// Mitsubishi GX Works2 project: Powder Spray robot1+ServoN   PLC: Q03UDV
// 20181022A

// task MAIN (event TRUE, interval 0, priority 31): MAIN
// task MAIN1 (event TRUE, interval 0, priority 31): MAIN1_Block000, MAIN1_Block001, MAIN1_Block002
// task OFS (event TRUE, interval 0, priority 31): OFS
// task LIFTER (event TRUE, interval 0, priority 31): LIFTER
// task 64AD (event TRUE, interval 0, priority 31): 64AD
// task SERVO (event TRUE, interval 0, priority 31): SERVO
// task D62 (event TRUE, interval 0, priority 31): D62
// task POWDER1 (event TRUE, interval 0, priority 31): POWDER1
// task POWDER2 (event TRUE, interval 0, priority 31): POWDER2
// task 62DA (event TRUE, interval 0, priority 31): 62DA

PROGRAM MAIN
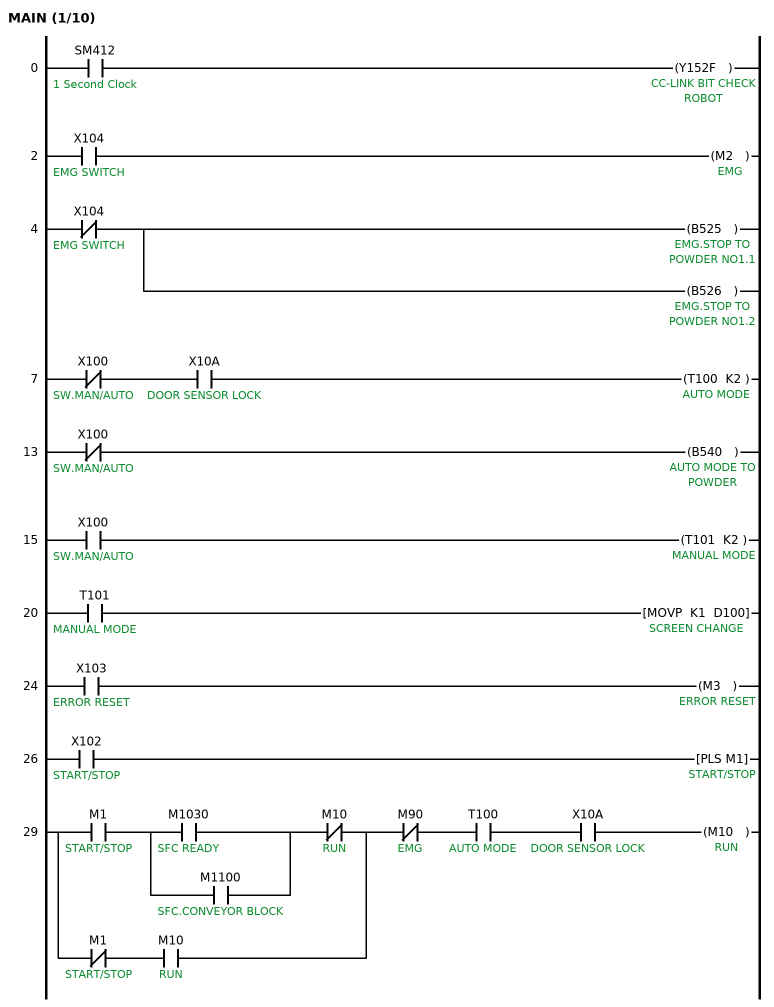
0     LD      SM412  ; 1 Second Clock
      OUT     Y152F  ; CC-LINK BIT CHECK ROBOT
2     LD      X104  ; EMG SWITCH
      OUT     M2  ; EMG
4     LDI     X104  ; EMG SWITCH
      OUT     B525  ; EMG.STOP TO POWDER NO1.1
      OUT     B526  ; EMG.STOP TO POWDER NO1.2
7     LDI     X100  ; SW.MAN/AUTO
      AND     X10A  ; DOOR SENSOR LOCK
      OUT     T100 K2  ; AUTO MODE
13    LDI     X100  ; SW.MAN/AUTO
      OUT     B540  ; AUTO MODE TO POWDER
15    LD      X100  ; SW.MAN/AUTO
      OUT     T101 K2  ; MANUAL MODE
20    LD      T101  ; MANUAL MODE
      MOVP    K1 D100  ; SCREEN CHANGE
24    LD      X103  ; ERROR RESET
      OUT     M3  ; ERROR RESET
26    LD      X102  ; START/STOP
      PLS     M1  ; START/STOP
29    LD      M1  ; START/STOP
      LD      M1030  ; SFC READY
      OR      M1100  ; SFC.CONVEYOR BLOCK
      ANB
      ANI     M10  ; RUN
      LDI     M1  ; START/STOP
      AND     M10  ; RUN
      ORB
      ANI     M90  ; EMG
      AND     T100  ; AUTO MODE
      AND     X10A  ; DOOR SENSOR LOCK
      OUT     M10  ; RUN
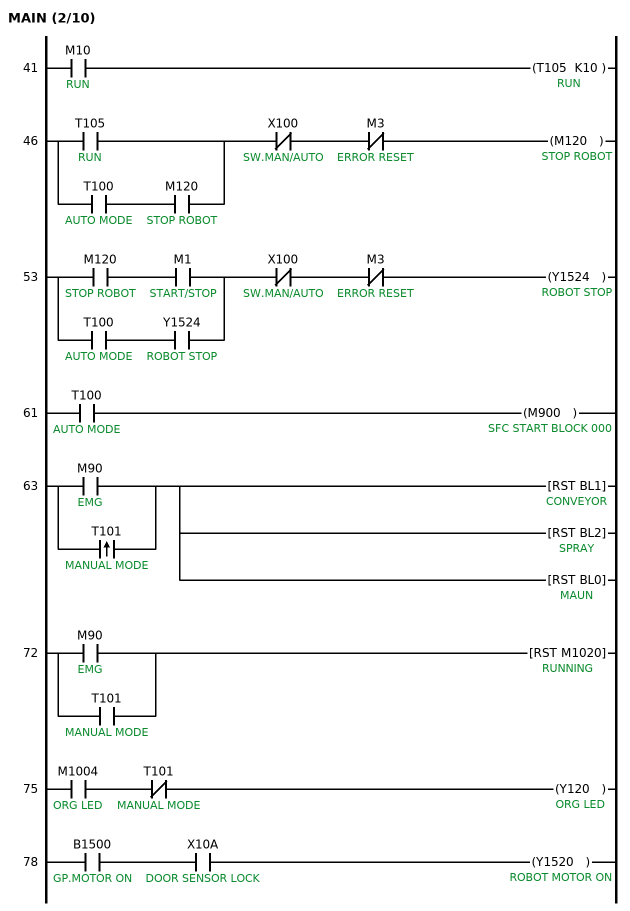
41    LD      M10  ; RUN
      OUT     T105 K10  ; RUN
46    LD      T105  ; RUN
      LD      T100  ; AUTO MODE
      AND     M120  ; STOP ROBOT
      ORB
      ANI     X100  ; SW.MAN/AUTO
      ANI     M3  ; ERROR RESET
      OUT     M120  ; STOP ROBOT
53    LD      M120  ; STOP ROBOT
      AND     M1  ; START/STOP
      LD      T100  ; AUTO MODE
      AND     Y1524  ; ROBOT STOP
      ORB
      ANI     X100  ; SW.MAN/AUTO
      ANI     M3  ; ERROR RESET
      OUT     Y1524  ; ROBOT STOP
61    LD      T100  ; AUTO MODE
      OUT     M900  ; SFC START BLOCK 000
63    LD      M90  ; EMG
      ORP     T101  ; MANUAL MODE
      RST     BL1  ; CONVEYOR
      RST     BL2  ; SPRAY
      RST     BL0  ; MAUN
72    LD      M90  ; EMG
      OR      T101  ; MANUAL MODE
      RST     M1020  ; RUNNING
75    LD      M1004  ; ORG LED
      ANI     T101  ; MANUAL MODE
      OUT     Y120  ; ORG LED
78    LD      B1500  ; GP.MOTOR ON
      AND     X10A  ; DOOR SENSOR LOCK
      OUT     Y1520  ; ROBOT MOTOR ON
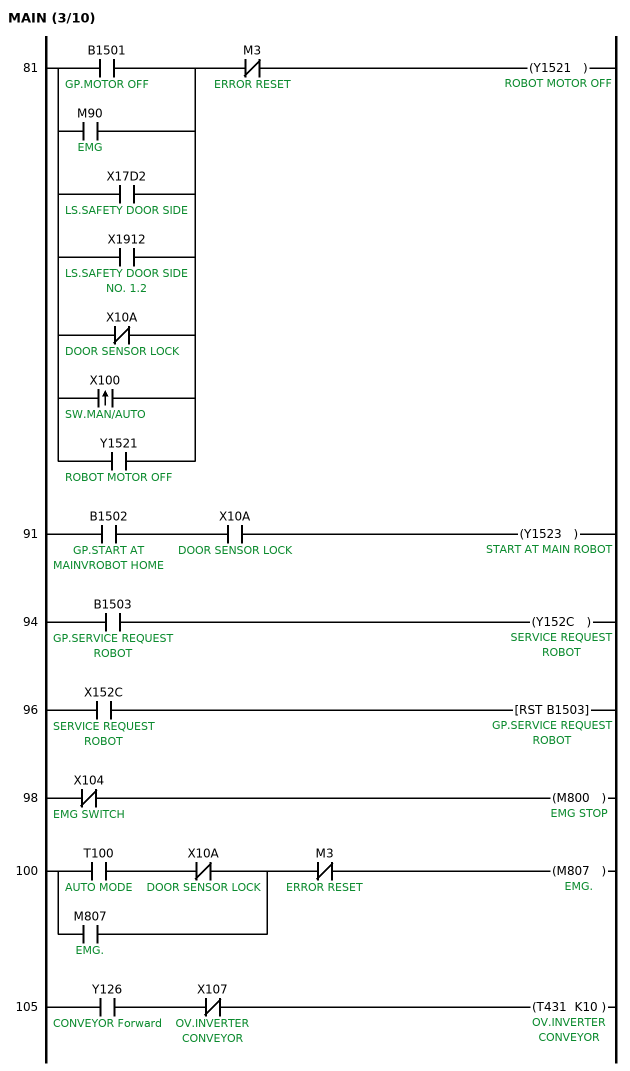
81    LD      B1501  ; GP.MOTOR OFF
      OR      M90  ; EMG
      OR      X17D2  ; LS.SAFETY DOOR SIDE
      OR      X1912  ; LS.SAFETY DOOR SIDE NO. 1.2
      ORI     X10A  ; DOOR SENSOR LOCK
      ORP     X100  ; SW.MAN/AUTO
      OR      Y1521  ; ROBOT MOTOR OFF
      ANI     M3  ; ERROR RESET
      OUT     Y1521  ; ROBOT MOTOR OFF
91    LD      B1502  ; GP.START AT MAINVROBOT HOME
      AND     X10A  ; DOOR SENSOR LOCK
      OUT     Y1523  ; START AT MAIN ROBOT
94    LD      B1503  ; GP.SERVICE REQUEST ROBOT
      OUT     Y152C  ; SERVICE REQUEST ROBOT
96    LD      X152C  ; SERVICE REQUEST ROBOT
      RST     B1503  ; GP.SERVICE REQUEST ROBOT
98    LDI     X104  ; EMG SWITCH
      OUT     M800  ; EMG STOP
100   LD      T100  ; AUTO MODE
      ANI     X10A  ; DOOR SENSOR LOCK
      OR      M807  ; EMG.
      ANI     M3  ; ERROR RESET
      OUT     M807  ; EMG.
105   LD      Y126  ; CONVEYOR Forward
      ANI     X107  ; OV.INVERTER CONVEYOR
      OUT     T431 K10  ; OV.INVERTER CONVEYOR
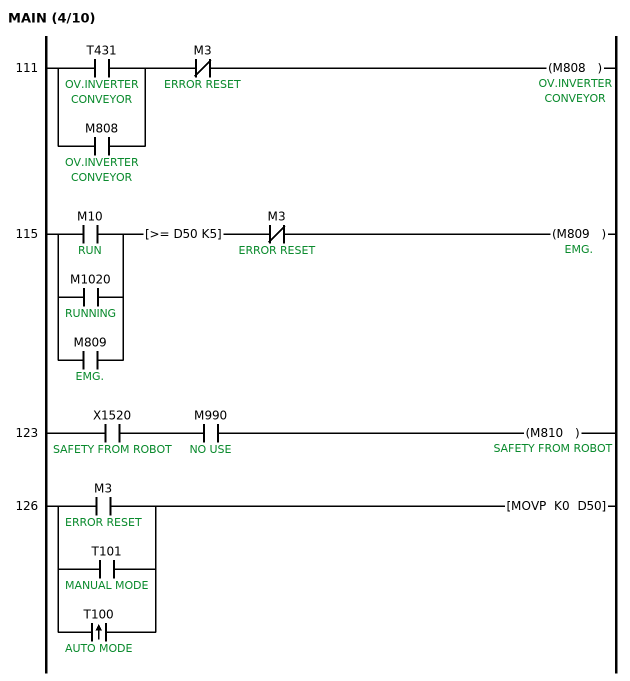
111   LD      T431  ; OV.INVERTER CONVEYOR
      OR      M808  ; OV.INVERTER CONVEYOR
      ANI     M3  ; ERROR RESET
      OUT     M808  ; OV.INVERTER CONVEYOR
115   LD      M10  ; RUN
      OR      M1020  ; RUNNING
      OR      M809  ; EMG.
      AND>=   D50 K5
      ANI     M3  ; ERROR RESET
      OUT     M809  ; EMG.
123   LD      X1520  ; SAFETY FROM ROBOT
      AND     M990  ; NO USE
      OUT     M810  ; SAFETY FROM ROBOT
126   LD      M3  ; ERROR RESET
      OR      T101  ; MANUAL MODE
      ORP     T100  ; AUTO MODE
      MOVP    K0 D50
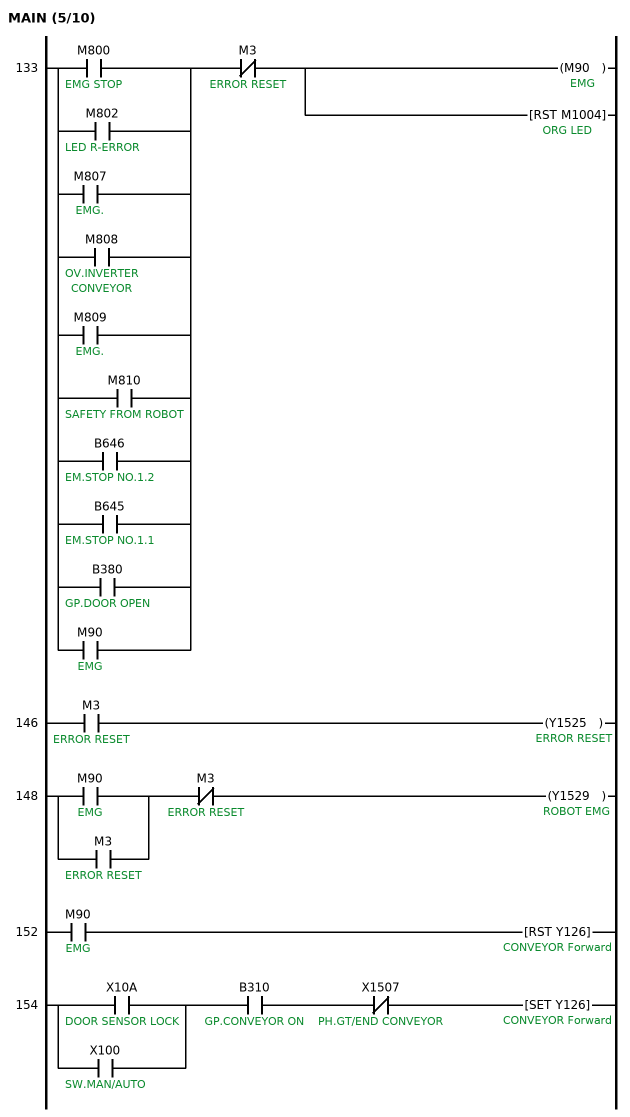
133   LD      M800  ; EMG STOP
      OR      M802  ; LED R-ERROR
      OR      M807  ; EMG.
      OR      M808  ; OV.INVERTER CONVEYOR
      OR      M809  ; EMG.
      OR      M810  ; SAFETY FROM ROBOT
      OR      B646  ; EM.STOP NO.1.2
      OR      B645  ; EM.STOP NO.1.1
      OR      B380  ; GP.DOOR OPEN
      OR      M90  ; EMG
      ANI     M3  ; ERROR RESET
      OUT     M90  ; EMG
      RST     M1004  ; ORG LED
146   LD      M3  ; ERROR RESET
      OUT     Y1525  ; ERROR RESET
148   LD      M90  ; EMG
      OR      M3  ; ERROR RESET
      ANI     M3  ; ERROR RESET
      OUT     Y1529  ; ROBOT EMG
152   LD      M90  ; EMG
      RST     Y126  ; CONVEYOR Forward
154   LD      X10A  ; DOOR SENSOR LOCK
      OR      X100  ; SW.MAN/AUTO
      AND     B310  ; GP.CONVEYOR ON
      ANI     X1507  ; PH.GT/END CONVEYOR
      SET     Y126  ; CONVEYOR Forward
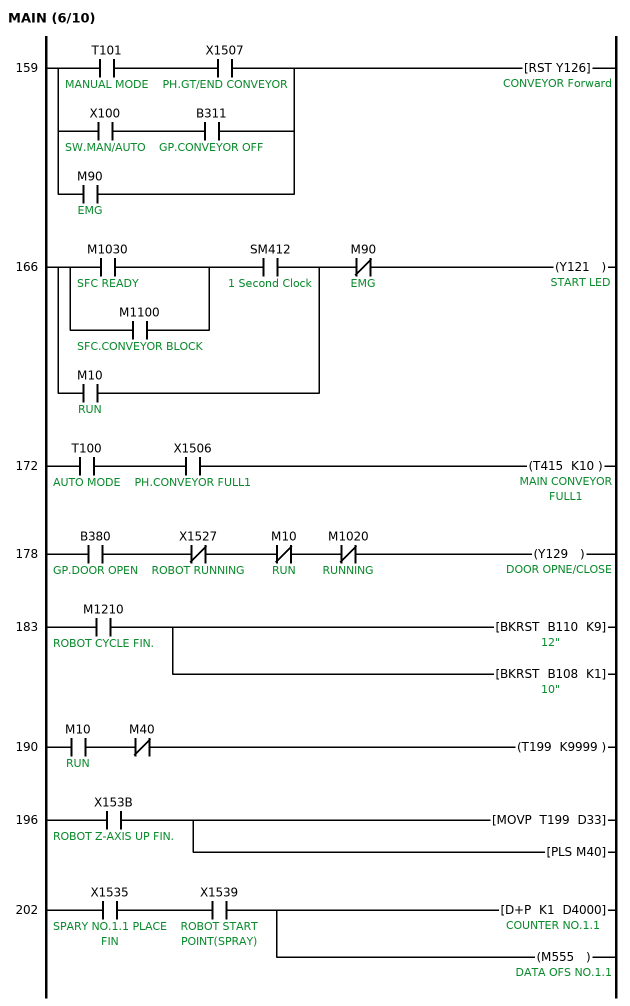
159   LD      T101  ; MANUAL MODE
      AND     X1507  ; PH.GT/END CONVEYOR
      LD      X100  ; SW.MAN/AUTO
      AND     B311  ; GP.CONVEYOR OFF
      ORB
      OR      M90  ; EMG
      RST     Y126  ; CONVEYOR Forward
166   LD      M1030  ; SFC READY
      OR      M1100  ; SFC.CONVEYOR BLOCK
      AND     SM412  ; 1 Second Clock
      OR      M10  ; RUN
      ANI     M90  ; EMG
      OUT     Y121  ; START LED
172   LD      T100  ; AUTO MODE
      AND     X1506  ; PH.CONVEYOR FULL1
      OUT     T415 K10  ; MAIN CONVEYOR FULL1
178   LD      B380  ; GP.DOOR OPEN
      ANI     X1527  ; ROBOT RUNNING
      ANI     M10  ; RUN
      ANI     M1020  ; RUNNING
      OUT     Y129  ; DOOR OPNE/CLOSE
183   LD      M1210  ; ROBOT CYCLE FIN.
      BKRST   B110 K9  ; 12"
      BKRST   B108 K1  ; 10"
190   LD      M10  ; RUN
      ANI     M40
      OUT     T199 K9999
196   LD      X153B  ; ROBOT Z-AXIS UP FIN.
      MOVP    T199 D33
      PLS     M40
202   LD      X1535  ; SPARY NO.1.1 PLACE FIN
      AND     X1539  ; ROBOT START POINT(SPRAY)
      D+P     K1 D4000  ; COUNTER NO.1.1
      OUT     M555  ; DATA OFS NO.1.1
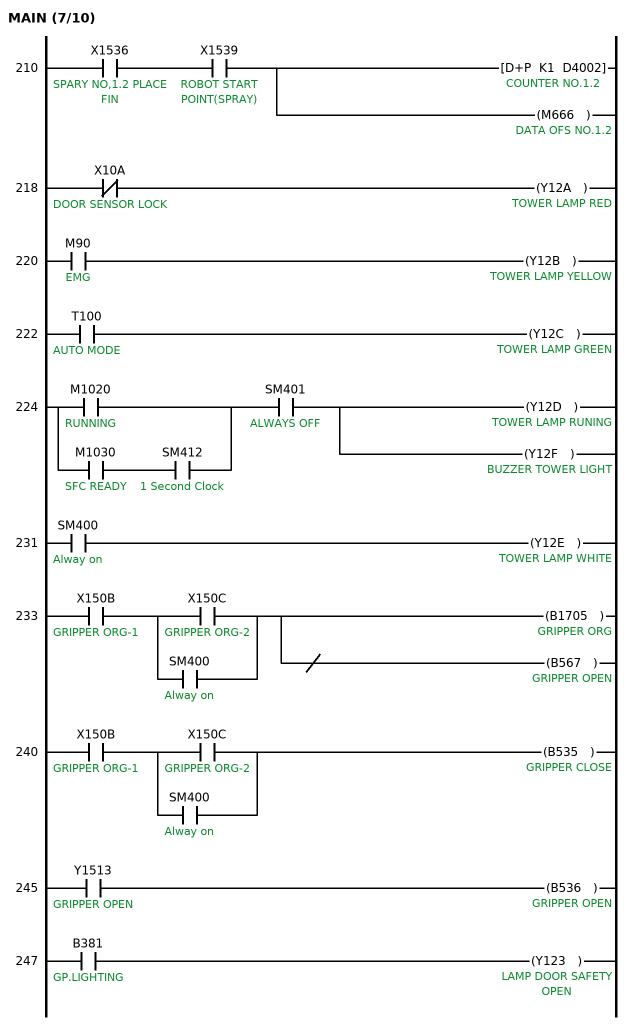
210   LD      X1536  ; SPARY NO,1.2 PLACE FIN
      AND     X1539  ; ROBOT START POINT(SPRAY)
      D+P     K1 D4002  ; COUNTER NO.1.2
      OUT     M666  ; DATA OFS NO.1.2
218   LDI     X10A  ; DOOR SENSOR LOCK
      OUT     Y12A  ; TOWER LAMP RED
220   LD      M90  ; EMG
      OUT     Y12B  ; TOWER LAMP YELLOW
222   LD      T100  ; AUTO MODE
      OUT     Y12C  ; TOWER LAMP GREEN
224   LD      M1020  ; RUNNING
      LD      M1030  ; SFC READY
      AND     SM412  ; 1 Second Clock
      ORB
      AND     SM401  ; ALWAYS OFF
      OUT     Y12D  ; TOWER LAMP RUNING
      OUT     Y12F  ; BUZZER TOWER LIGHT
231   LD      SM400  ; Alway on
      OUT     Y12E  ; TOWER LAMP WHITE
233   LD      X150B  ; GRIPPER ORG-1
      LD      X150C  ; GRIPPER ORG-2
      OR      SM400  ; Alway on
      ANB
      OUT     B1705  ; GRIPPER ORG
      INV
      OUT     B567  ; GRIPPER OPEN
240   LD      X150B  ; GRIPPER ORG-1
      LD      X150C  ; GRIPPER ORG-2
      OR      SM400  ; Alway on
      ANB
      OUT     B535  ; GRIPPER CLOSE
245   LD      Y1513  ; GRIPPER OPEN
      OUT     B536  ; GRIPPER OPEN
247   LD      B381  ; GP.LIGHTING
      OUT     Y123  ; LAMP DOOR SAFETY OPEN
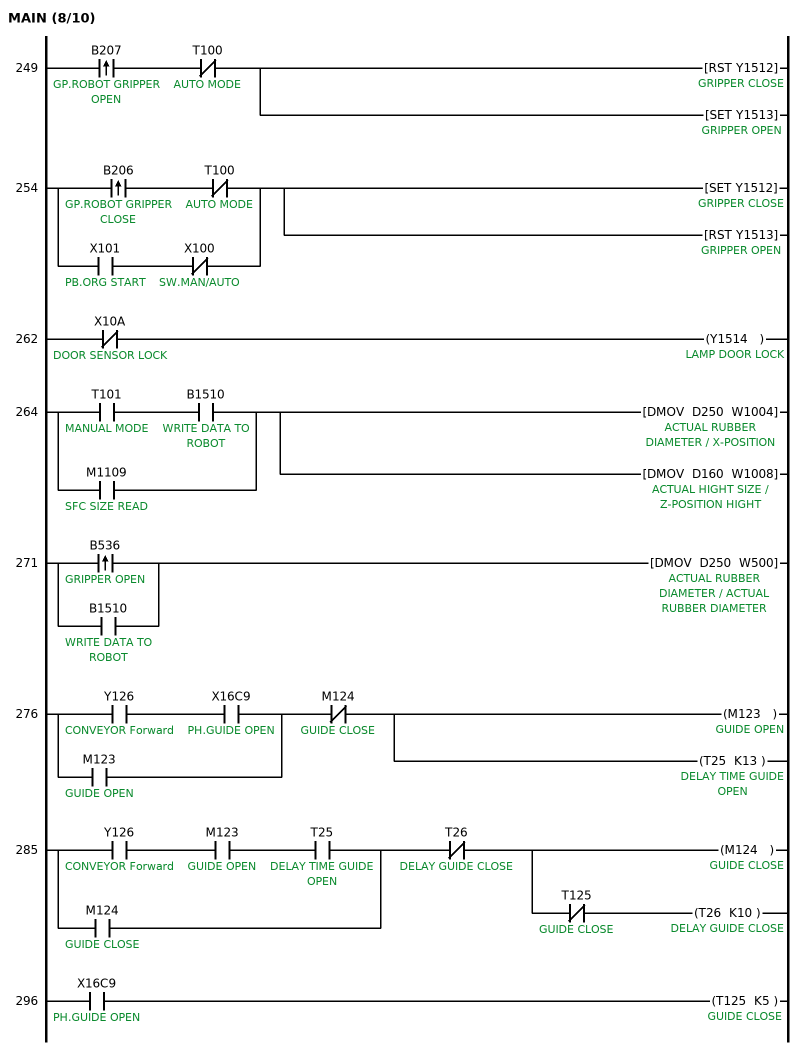
249   LDP     B207  ; GP.ROBOT GRIPPER OPEN
      ANI     T100  ; AUTO MODE
      RST     Y1512  ; GRIPPER CLOSE
      SET     Y1513  ; GRIPPER OPEN
254   LDP     B206  ; GP.ROBOT GRIPPER CLOSE
      ANI     T100  ; AUTO MODE
      LD      X101  ; PB.ORG START
      ANI     X100  ; SW.MAN/AUTO
      ORB
      SET     Y1512  ; GRIPPER CLOSE
      RST     Y1513  ; GRIPPER OPEN
262   LDI     X10A  ; DOOR SENSOR LOCK
      OUT     Y1514  ; LAMP DOOR LOCK
264   LD      T101  ; MANUAL MODE
      AND     B1510  ; WRITE DATA TO ROBOT
      OR      M1109  ; SFC SIZE READ
      DMOV    D250 W1004  ; ACTUAL RUBBER DIAMETER / X-POSITION
      DMOV    D160 W1008  ; ACTUAL HIGHT SIZE / Z-POSITION HIGHT
271   LDP     B536  ; GRIPPER OPEN
      OR      B1510  ; WRITE DATA TO ROBOT
      DMOV    D250 W500  ; ACTUAL RUBBER DIAMETER
276   LD      Y126  ; CONVEYOR Forward
      AND     X16C9  ; PH.GUIDE OPEN
      OR      M123  ; GUIDE OPEN
      ANI     M124  ; GUIDE CLOSE
      OUT     M123  ; GUIDE OPEN
      OUT     T25 K13  ; DELAY TIME GUIDE OPEN
285   LD      Y126  ; CONVEYOR Forward
      AND     M123  ; GUIDE OPEN
      AND     T25  ; DELAY TIME GUIDE OPEN
      OR      M124  ; GUIDE CLOSE
      ANI     T26  ; DELAY GUIDE CLOSE
      OUT     M124  ; GUIDE CLOSE
      ANI     T125  ; GUIDE CLOSE
      OUT     T26 K10  ; DELAY GUIDE CLOSE
296   LD      X16C9  ; PH.GUIDE OPEN
      OUT     T125 K5  ; GUIDE CLOSE
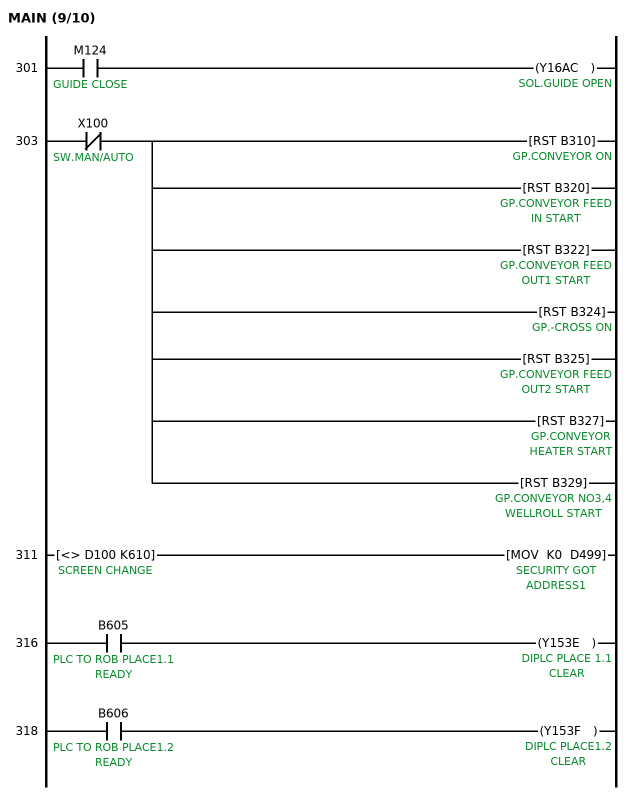
301   LD      M124  ; GUIDE CLOSE
      OUT     Y16AC  ; SOL.GUIDE OPEN
303   LDI     X100  ; SW.MAN/AUTO
      RST     B310  ; GP.CONVEYOR ON
      RST     B320  ; GP.CONVEYOR FEED IN START
      RST     B322  ; GP.CONVEYOR FEED OUT1 START
      RST     B324  ; GP.-CROSS ON
      RST     B325  ; GP.CONVEYOR FEED OUT2 START
      RST     B327  ; GP.CONVEYOR HEATER START
      RST     B329  ; GP.CONVEYOR NO3,4 WELLROLL START
311   LD<>    D100 K610  ; SCREEN CHANGE
      MOV     K0 D499  ; SECURITY GOT ADDRESS1
316   LD      B605  ; PLC TO ROB PLACE1.1 READY
      OUT     Y153E  ; DIPLC PLACE 1.1 CLEAR
318   LD      B606  ; PLC TO ROB PLACE1.2 READY
      OUT     Y153F  ; DIPLC PLACE1.2  CLEAR
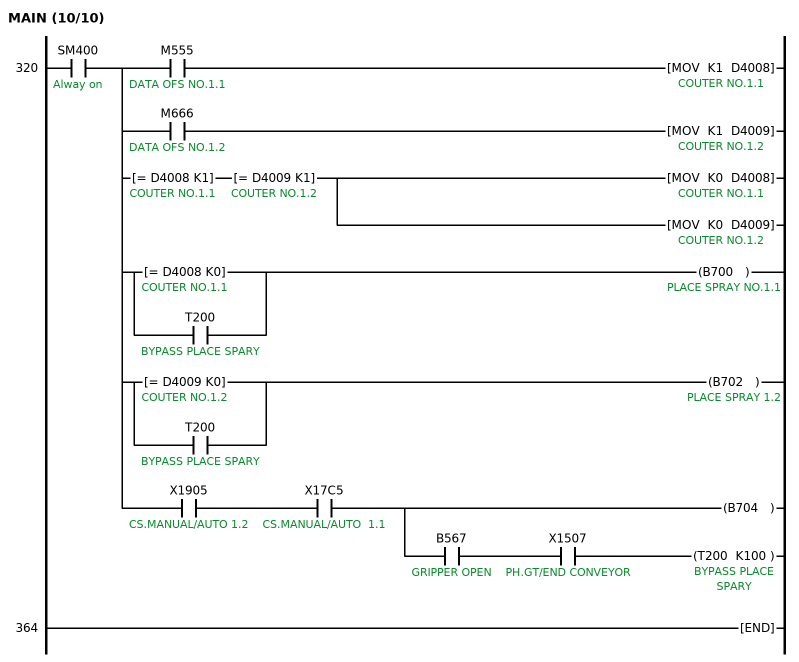
320   LD      SM400  ; Alway on
      MPS
      AND     M555  ; DATA OFS NO.1.1
      MOV     K1 D4008  ; COUTER NO.1.1
      MRD
      AND     M666  ; DATA OFS NO.1.2
      MOV     K1 D4009  ; COUTER NO.1.2
      MRD
      AND=    D4008 K1  ; COUTER NO.1.1
      AND=    D4009 K1  ; COUTER NO.1.2
      MOV     K0 D4008
      MOV     K0 D4009
      MRD
      LD=     D4008 K0  ; COUTER NO.1.1
      OR      T200  ; BYPASS PLACE SPARY
      ANB
      OUT     B700  ; PLACE SPRAY NO.1.1
      MRD
      LD=     D4009 K0  ; COUTER NO.1.2
      OR      T200  ; BYPASS PLACE SPARY
      ANB
      OUT     B702  ; PLACE SPRAY 1.2
      MPP
      AND     X1905  ; CS.MANUAL/AUTO 1.2
      AND     X17C5  ; CS.MANUAL/AUTO  1.1
      OUT     B704
      AND     B567  ; GRIPPER OPEN
      AND     X1507  ; PH.GT/END CONVEYOR
      OUT     T200 K100  ; BYPASS PLACE SPARY
364   END
END_PROGRAM

PROGRAM OFS
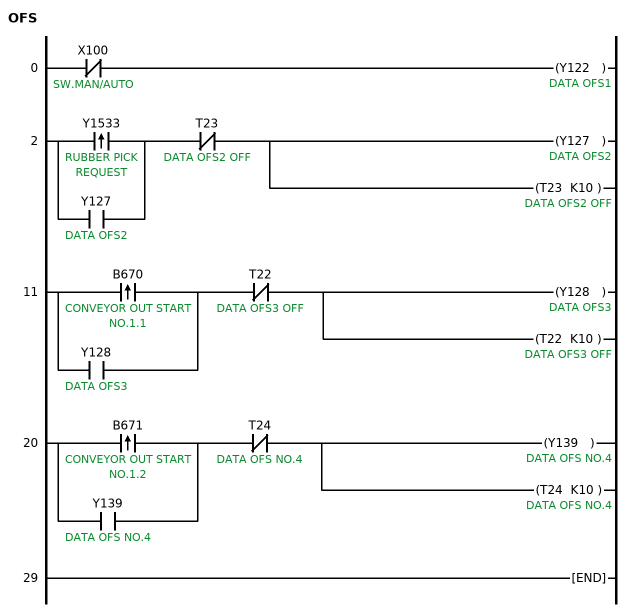
0     LDI     X100  ; SW.MAN/AUTO
      OUT     Y122  ; DATA OFS1
2     LDP     Y1533  ; RUBBER PICK  REQUEST
      OR      Y127  ; DATA OFS2
      ANI     T23  ; DATA OFS2 OFF
      OUT     Y127  ; DATA OFS2
      OUT     T23 K10  ; DATA OFS2 OFF
11    LDP     B670  ; CONVEYOR OUT START NO.1.1
      OR      Y128  ; DATA OFS3
      ANI     T22  ; DATA OFS3 OFF
      OUT     Y128  ; DATA OFS3
      OUT     T22 K10  ; DATA OFS3 OFF
20    LDP     B671  ; CONVEYOR OUT START NO.1.2
      OR      Y139  ; DATA OFS NO.4
      ANI     T24  ; DATA OFS NO.4
      OUT     Y139  ; DATA OFS NO.4
      OUT     T24 K10  ; DATA OFS NO.4
29    END
END_PROGRAM

PROGRAM LIFTER
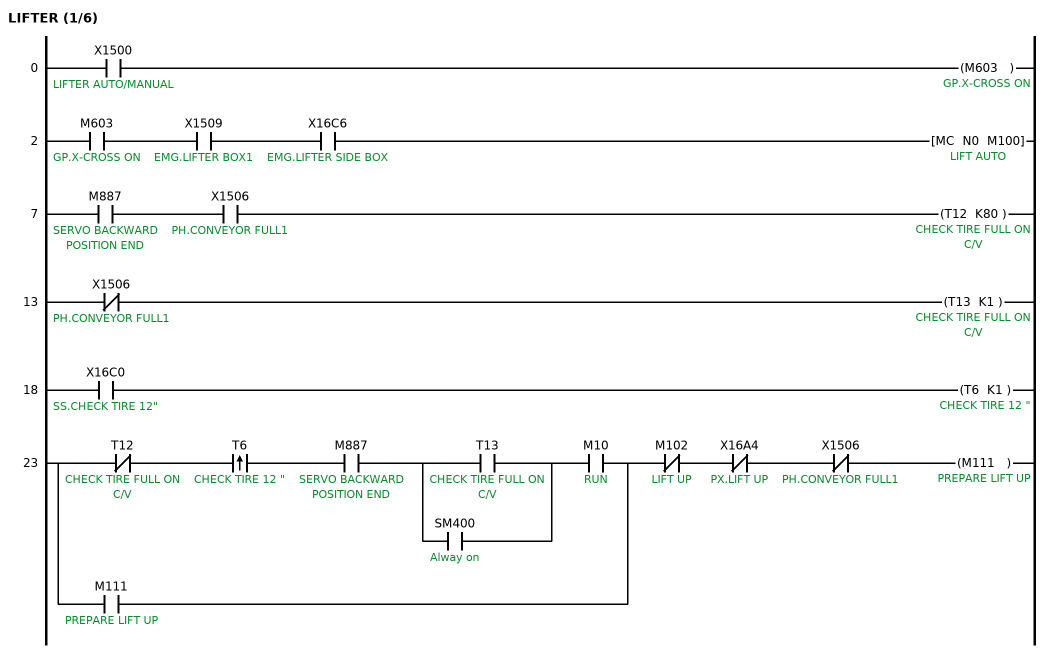
0     LD      X1500  ; LIFTER AUTO/MANUAL
      OUT     M603  ; GP.X-CROSS ON
2     LD      M603  ; GP.X-CROSS ON
      AND     X1509  ; EMG.LIFTER BOX1
      AND     X16C6  ; EMG.LIFTER SIDE BOX
      MC      N0 M100  ; LIFT AUTO
7     LD      M887  ; SERVO BACKWARD POSITION END
      AND     X1506  ; PH.CONVEYOR FULL1
      OUT     T12 K80  ; CHECK TIRE FULL ON C/V
13    LDI     X1506  ; PH.CONVEYOR FULL1
      OUT     T13 K1  ; CHECK TIRE FULL ON C/V
18    LD      X16C0  ; SS.CHECK TIRE 12"
      OUT     T6 K1  ; CHECK TIRE 12 "
23    LDI     T12  ; CHECK TIRE FULL ON C/V
      ANDP    T6  ; CHECK TIRE 12 "
      AND     M887  ; SERVO BACKWARD POSITION END
      LD      T13  ; CHECK TIRE FULL ON C/V
      OR      SM400  ; Alway on
      ANB
      AND     M10  ; RUN
      OR      M111  ; PREPARE LIFT UP
      ANI     M102  ; LIFT UP
      ANI     X16A4  ; PX.LIFT UP
      ANI     X1506  ; PH.CONVEYOR FULL1
      OUT     M111  ; PREPARE LIFT UP
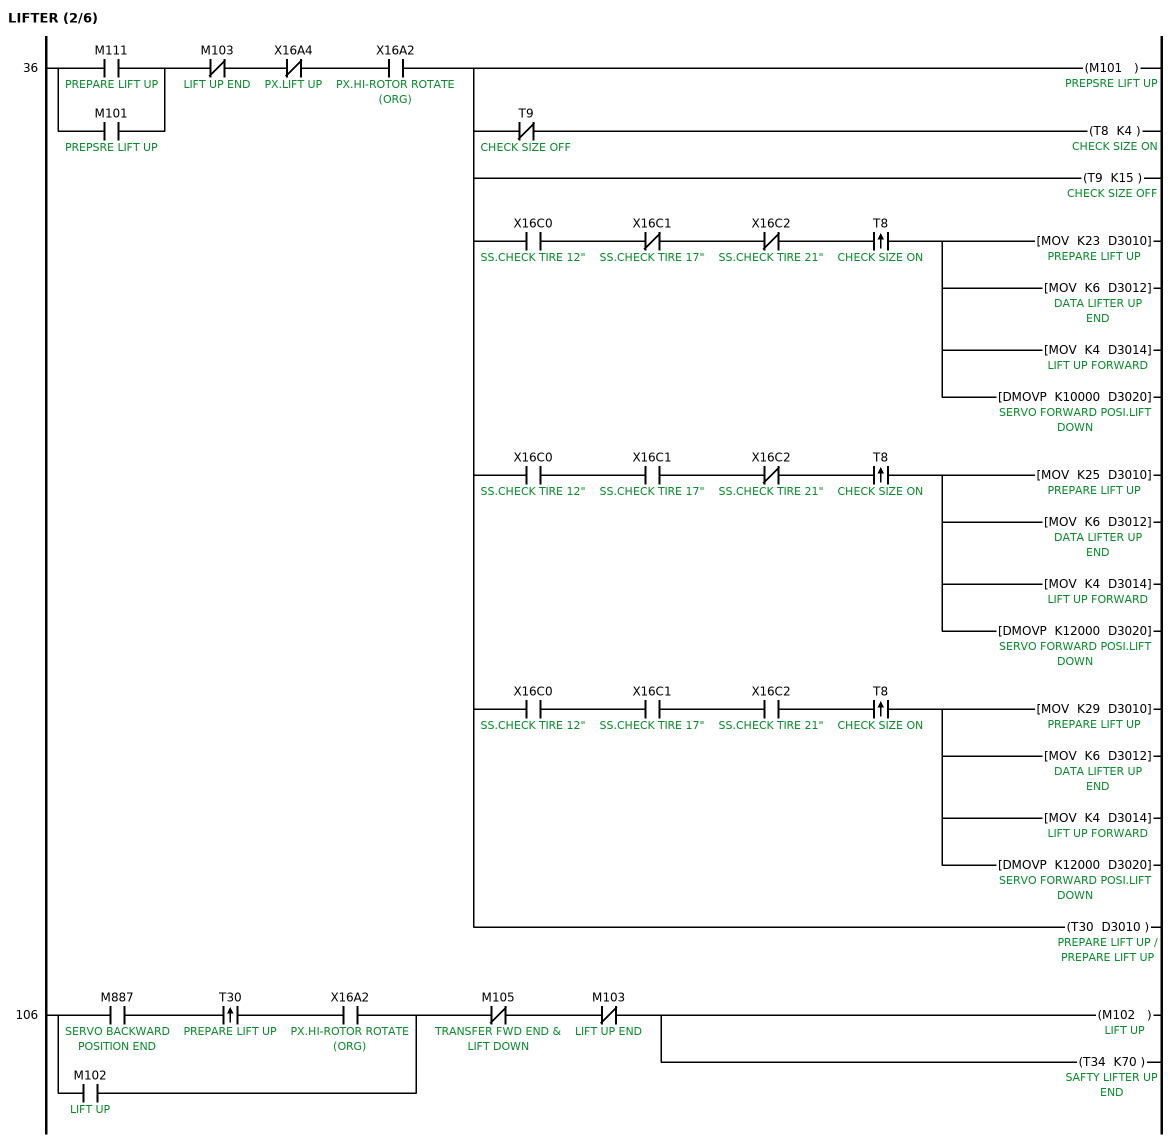
36    LD      M111  ; PREPARE LIFT UP
      OR      M101  ; PREPSRE LIFT UP
      ANI     M103  ; LIFT UP END
      ANI     X16A4  ; PX.LIFT UP
      AND     X16A2  ; PX.HI-ROTOR ROTATE (ORG)
      OUT     M101  ; PREPSRE LIFT UP
      MPS
      ANI     T9  ; CHECK SIZE OFF
      OUT     T8 K4  ; CHECK SIZE ON
      MPP
      OUT     T9 K15  ; CHECK SIZE OFF
      MPS
      AND     X16C0  ; SS.CHECK TIRE 12"
      ANI     X16C1  ; SS.CHECK TIRE 17"
      ANI     X16C2  ; SS.CHECK TIRE 21"
      ANDP    T8  ; CHECK SIZE ON
      MOV     K23 D3010  ; PREPARE LIFT UP
      MOV     K6 D3012  ; DATA LIFTER UP  END
      MOV     K4 D3014  ; LIFT UP FORWARD
      DMOVP   K10000 D3020  ; SERVO FORWARD POSI.LIFT DOWN
      MRD
      AND     X16C0  ; SS.CHECK TIRE 12"
      AND     X16C1  ; SS.CHECK TIRE 17"
      ANI     X16C2  ; SS.CHECK TIRE 21"
      ANDP    T8  ; CHECK SIZE ON
      MOV     K25 D3010
      MOV     K6 D3012
      MOV     K4 D3014
      DMOVP   K12000 D3020
      MRD
      AND     X16C0  ; SS.CHECK TIRE 12"
      AND     X16C1  ; SS.CHECK TIRE 17"
      AND     X16C2  ; SS.CHECK TIRE 21"
      ANDP    T8  ; CHECK SIZE ON
      MOV     K29 D3010
      MOV     K6 D3012
      MOV     K4 D3014
      DMOVP   K12000 D3020
      MPP
      OUT     T30 D3010  ; PREPARE LIFT UP / PREPARE LIFT UP
106   LD      M887  ; SERVO BACKWARD POSITION END
      ANDP    T30  ; PREPARE LIFT UP
      AND     X16A2  ; PX.HI-ROTOR ROTATE (ORG)
      OR      M102  ; LIFT UP
      ANI     M105  ; TRANSFER FWD END & LIFT DOWN
      ANI     M103  ; LIFT UP END
      OUT     M102  ; LIFT UP
      OUT     T34 K70  ; SAFTY LIFTER UP END
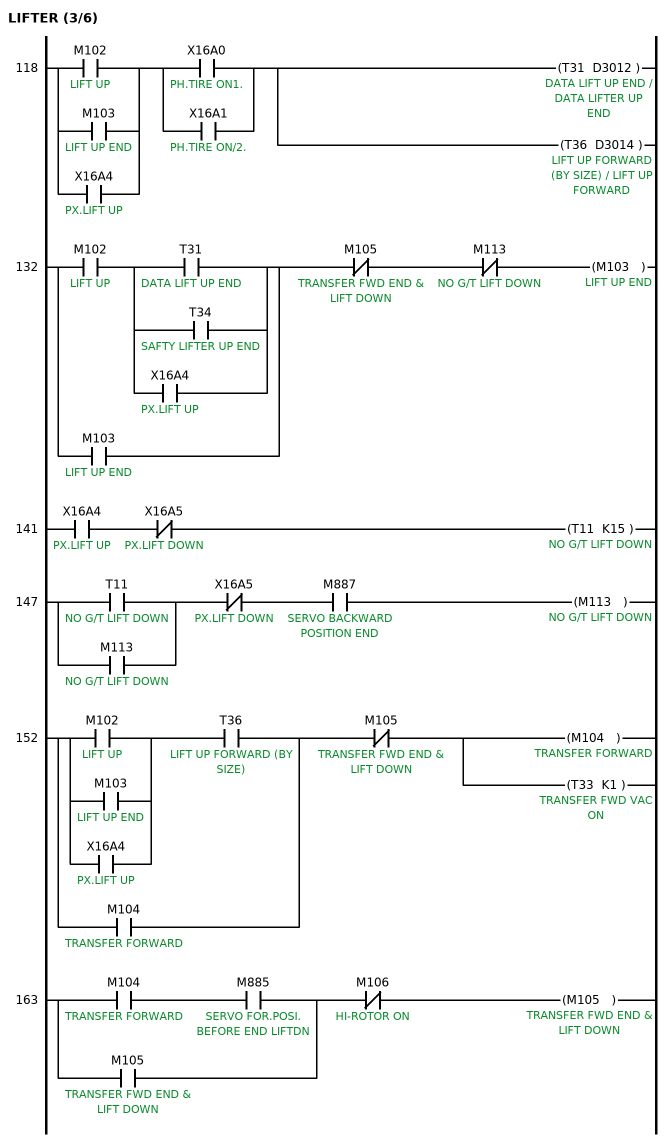
118   LD      M102  ; LIFT UP
      OR      M103  ; LIFT UP END
      OR      X16A4  ; PX.LIFT UP
      LD      X16A0  ; PH.TIRE ON1.
      OR      X16A1  ; PH.TIRE ON/2.
      ANB
      OUT     T31 D3012  ; DATA LIFT UP END / DATA LIFTER UP  END
      OUT     T36 D3014  ; LIFT UP FORWARD (BY SIZE) / LIFT UP FORWARD
132   LD      M102  ; LIFT UP
      LD      T31  ; DATA LIFT UP END
      OR      T34  ; SAFTY LIFTER UP END
      OR      X16A4  ; PX.LIFT UP
      ANB
      OR      M103  ; LIFT UP END
      ANI     M105  ; TRANSFER FWD END & LIFT DOWN
      ANI     M113  ; NO G/T LIFT DOWN
      OUT     M103  ; LIFT UP END
141   LD      X16A4  ; PX.LIFT UP
      ANI     X16A5  ; PX.LIFT DOWN
      OUT     T11 K15  ; NO G/T LIFT DOWN
147   LD      T11  ; NO G/T LIFT DOWN
      OR      M113  ; NO G/T LIFT DOWN
      ANI     X16A5  ; PX.LIFT DOWN
      AND     M887  ; SERVO BACKWARD POSITION END
      OUT     M113  ; NO G/T LIFT DOWN
152   LD      M102  ; LIFT UP
      OR      M103  ; LIFT UP END
      OR      X16A4  ; PX.LIFT UP
      AND     T36  ; LIFT UP FORWARD (BY SIZE)
      OR      M104  ; TRANSFER FORWARD
      ANI     M105  ; TRANSFER FWD END & LIFT DOWN
      OUT     M104  ; TRANSFER FORWARD
      OUT     T33 K1  ; TRANSFER FWD VAC ON
163   LD      M104  ; TRANSFER FORWARD
      AND     M885  ; SERVO FOR.POSI.BEFORE END LIFTDN
      OR      M105  ; TRANSFER FWD END & LIFT DOWN
      ANI     M106  ; HI-ROTOR ON
      OUT     M105  ; TRANSFER FWD END & LIFT DOWN
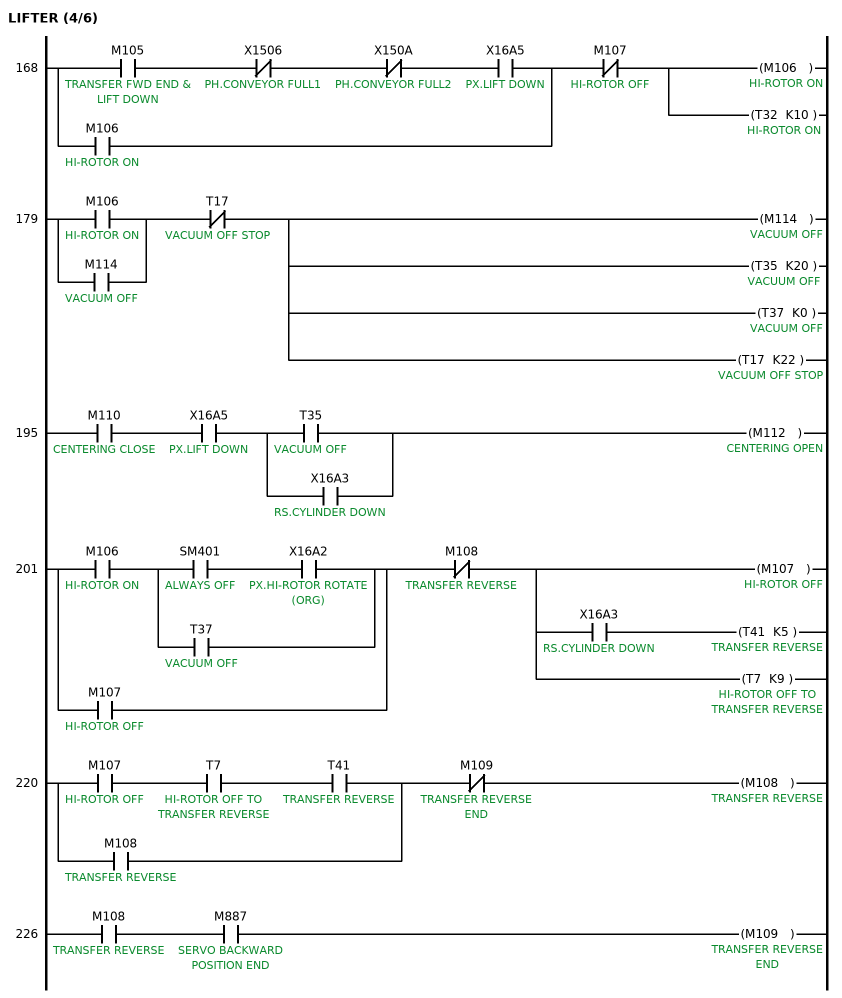
168   LD      M105  ; TRANSFER FWD END & LIFT DOWN
      ANI     X1506  ; PH.CONVEYOR FULL1
      ANI     X150A  ; PH.CONVEYOR FULL2
      AND     X16A5  ; PX.LIFT DOWN
      OR      M106  ; HI-ROTOR ON
      ANI     M107  ; HI-ROTOR OFF
      OUT     M106  ; HI-ROTOR ON
      OUT     T32 K10  ; HI-ROTOR ON
179   LD      M106  ; HI-ROTOR ON
      OR      M114  ; VACUUM OFF
      ANI     T17  ; VACUUM OFF STOP
      OUT     M114  ; VACUUM OFF
      OUT     T35 K20  ; VACUUM OFF
      OUT     T37 K0  ; VACUUM OFF
      OUT     T17 K22  ; VACUUM OFF STOP
195   LD      M110  ; CENTERING CLOSE
      AND     X16A5  ; PX.LIFT DOWN
      LD      T35  ; VACUUM OFF
      OR      X16A3  ; RS.CYLINDER DOWN
      ANB
      OUT     M112  ; CENTERING OPEN
201   LD      M106  ; HI-ROTOR ON
      LD      SM401  ; ALWAYS OFF
      AND     X16A2  ; PX.HI-ROTOR ROTATE (ORG)
      OR      T37  ; VACUUM OFF
      ANB
      OR      M107  ; HI-ROTOR OFF
      ANI     M108  ; TRANSFER REVERSE
      OUT     M107  ; HI-ROTOR OFF
      MPS
      AND     X16A3  ; RS.CYLINDER DOWN
      OUT     T41 K5  ; TRANSFER REVERSE
      MPP
      OUT     T7 K9  ; HI-ROTOR OFF TO TRANSFER REVERSE
220   LD      M107  ; HI-ROTOR OFF
      AND     T7  ; HI-ROTOR OFF TO TRANSFER REVERSE
      AND     T41  ; TRANSFER REVERSE
      OR      M108  ; TRANSFER REVERSE
      ANI     M109  ; TRANSFER REVERSE END
      OUT     M108  ; TRANSFER REVERSE
226   LD      M108  ; TRANSFER REVERSE
      AND     M887  ; SERVO BACKWARD POSITION END
      OUT     M109  ; TRANSFER REVERSE END
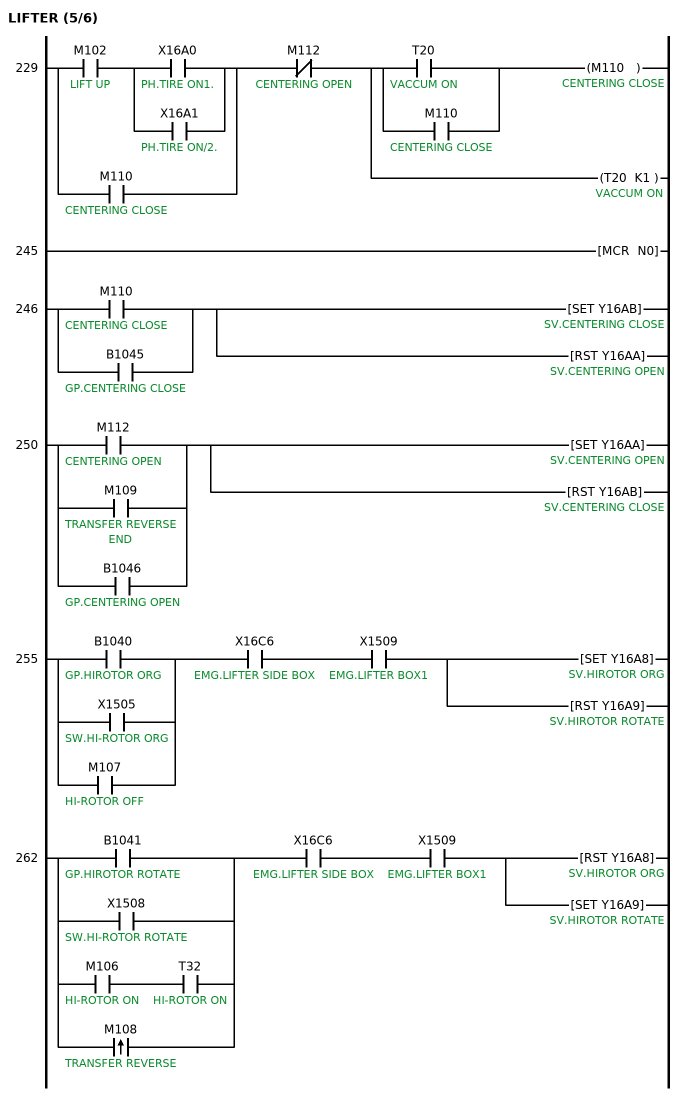
229   LD      M102  ; LIFT UP
      LD      X16A0  ; PH.TIRE ON1.
      OR      X16A1  ; PH.TIRE ON/2.
      ANB
      OR      M110  ; CENTERING CLOSE
      ANI     M112  ; CENTERING OPEN
      MPS
      LD      T20  ; VACCUM ON
      OR      M110  ; CENTERING CLOSE
      ANB
      OUT     M110  ; CENTERING CLOSE
      MPP
      OUT     T20 K1  ; VACCUM ON
245   MCR     N0
246   LD      M110  ; CENTERING CLOSE
      OR      B1045  ; GP.CENTERING CLOSE
      SET     Y16AB  ; SV.CENTERING CLOSE
      RST     Y16AA  ; SV.CENTERING OPEN
250   LD      M112  ; CENTERING OPEN
      OR      M109  ; TRANSFER REVERSE END
      OR      B1046  ; GP.CENTERING OPEN
      SET     Y16AA  ; SV.CENTERING OPEN
      RST     Y16AB  ; SV.CENTERING CLOSE
255   LD      B1040  ; GP.HIROTOR ORG
      OR      X1505  ; SW.HI-ROTOR ORG
      OR      M107  ; HI-ROTOR OFF
      AND     X16C6  ; EMG.LIFTER SIDE BOX
      AND     X1509  ; EMG.LIFTER BOX1
      SET     Y16A8  ; SV.HIROTOR ORG
      RST     Y16A9  ; SV.HIROTOR ROTATE
262   LD      B1041  ; GP.HIROTOR ROTATE
      OR      X1508  ; SW.HI-ROTOR ROTATE
      LD      M106  ; HI-ROTOR ON
      AND     T32  ; HI-ROTOR ON
      ORB
      ORP     M108  ; TRANSFER REVERSE
      AND     X16C6  ; EMG.LIFTER SIDE BOX
      AND     X1509  ; EMG.LIFTER BOX1
      RST     Y16A8  ; SV.HIROTOR ORG
      SET     Y16A9  ; SV.HIROTOR ROTATE
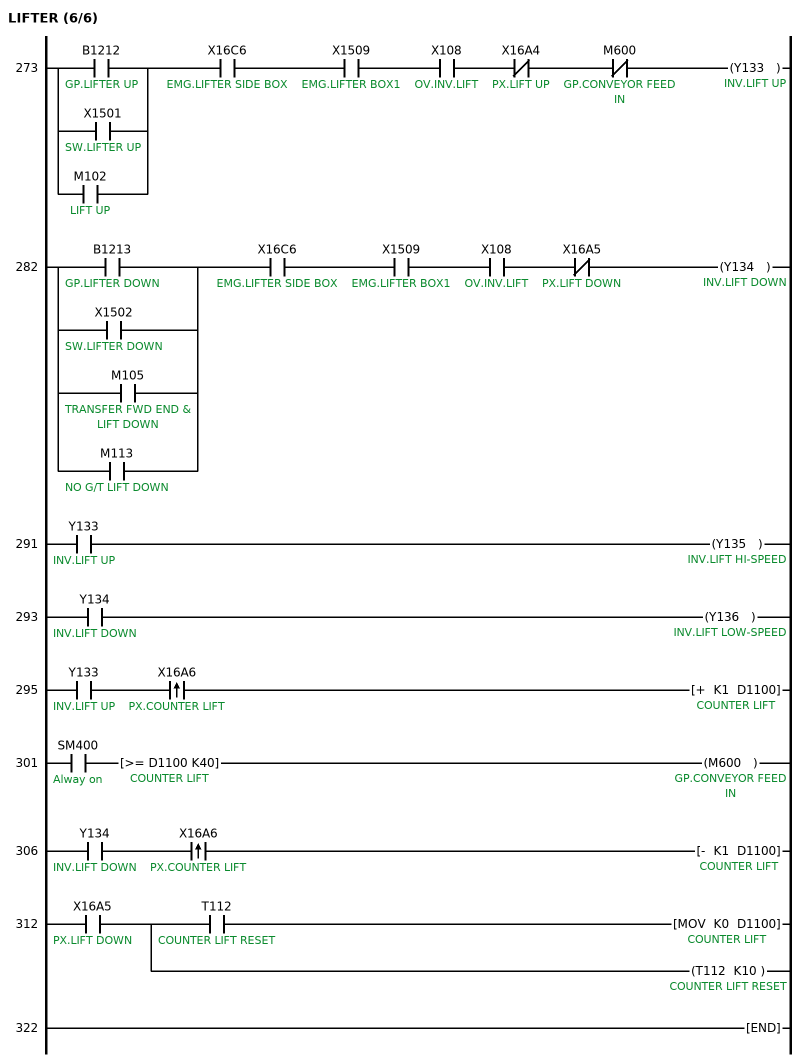
273   LD      B1212  ; GP.LIFTER UP
      OR      X1501  ; SW.LIFTER UP
      OR      M102  ; LIFT UP
      AND     X16C6  ; EMG.LIFTER SIDE BOX
      AND     X1509  ; EMG.LIFTER BOX1
      AND     X108  ; OV.INV.LIFT
      ANI     X16A4  ; PX.LIFT UP
      ANI     M600  ; GP.CONVEYOR FEED IN
      OUT     Y133  ; INV.LIFT UP
282   LD      B1213  ; GP.LIFTER DOWN
      OR      X1502  ; SW.LIFTER DOWN
      OR      M105  ; TRANSFER FWD END & LIFT DOWN
      OR      M113  ; NO G/T LIFT DOWN
      AND     X16C6  ; EMG.LIFTER SIDE BOX
      AND     X1509  ; EMG.LIFTER BOX1
      AND     X108  ; OV.INV.LIFT
      ANI     X16A5  ; PX.LIFT DOWN
      OUT     Y134  ; INV.LIFT DOWN
291   LD      Y133  ; INV.LIFT UP
      OUT     Y135  ; INV.LIFT HI-SPEED
293   LD      Y134  ; INV.LIFT DOWN
      OUT     Y136  ; INV.LIFT LOW-SPEED
295   LD      Y133  ; INV.LIFT UP
      ANDP    X16A6  ; PX.COUNTER LIFT
      +       K1 D1100  ; COUNTER LIFT
301   LD      SM400  ; Alway on
      AND>=   D1100 K40  ; COUNTER LIFT
      OUT     M600  ; GP.CONVEYOR FEED IN
306   LD      Y134  ; INV.LIFT DOWN
      ANDP    X16A6  ; PX.COUNTER LIFT
      -       K1 D1100
312   LD      X16A5  ; PX.LIFT DOWN
      MPS
      AND     T112  ; COUNTER LIFT RESET
      MOV     K0 D1100
      MPP
      OUT     T112 K10  ; COUNTER LIFT RESET
322   END
END_PROGRAM

PROGRAM 64AD
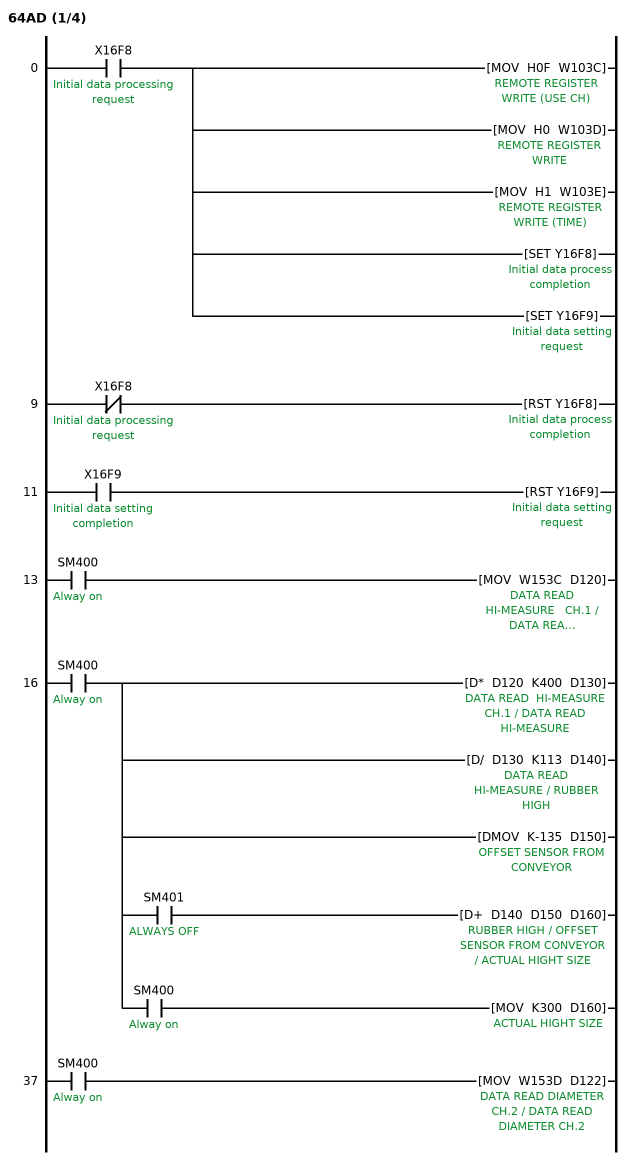
0     LD      X16F8  ; Initial data processing request
      MOV     H0F W103C  ; REMOTE REGISTER WRITE (USE CH)
      MOV     H0 W103D  ; REMOTE REGISTER WRITE
      MOV     H1 W103E  ; REMOTE REGISTER WRITE (TIME)
      SET     Y16F8  ; Initial data process completion
      SET     Y16F9  ; Initial data setting request
9     LDI     X16F8  ; Initial data processing request
      RST     Y16F8  ; Initial data process completion
11    LD      X16F9  ; Initial data setting completion
      RST     Y16F9  ; Initial data setting request
13    LD      SM400  ; Alway on
      MOV     W153C D120  ; DATA READ  HI-MEASURE   CH.1 / DATA READ  HI-MEASURE CH.1
16    LD      SM400  ; Alway on
      D*      D120 K400 D130  ; DATA READ  HI-MEASURE
      D/      D130 K113 D140  ; RUBBER HIGH
      DMOV    K-135 D150  ; OFFSET SENSOR FROM CONVEYOR
      MPS
      AND     SM401  ; ALWAYS OFF
      D+      D140 D150 D160  ; ACTUAL HIGHT SIZE
      MPP
      AND     SM400  ; Alway on
      MOV     K300 D160
37    LD      SM400  ; Alway on
      MOV     W153D D122  ; DATA READ DIAMETER CH.2 / DATA READ DIAMETER CH.2
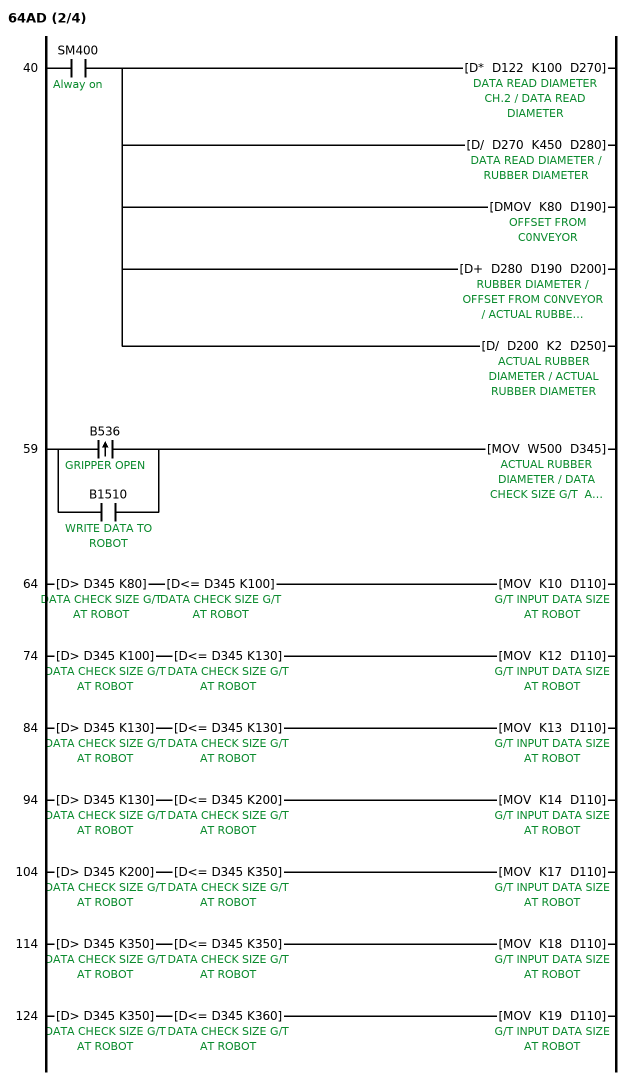
40    LD      SM400  ; Alway on
      D*      D122 K100 D270  ; DATA READ DIAMETER
      D/      D270 K450 D280  ; RUBBER DIAMETER
      DMOV    K80 D190  ; OFFSET FROM C0NVEYOR
      D+      D280 D190 D200  ; ACTUAL RUBBER DIAMETER
      D/      D200 K2 D250  ; ACTUAL RUBBER DIAMETER
59    LDP     B536  ; GRIPPER OPEN
      OR      B1510  ; WRITE DATA TO ROBOT
      MOV     W500 D345  ; ACTUAL RUBBER DIAMETER / DATA CHECK SIZE G/T  AT ROBOT
64    LDD>    D345 K80  ; DATA CHECK SIZE G/T  AT ROBOT
      ANDD<=  D345 K100  ; DATA CHECK SIZE G/T  AT ROBOT
      MOV     K10 D110  ; G/T INPUT DATA SIZE AT ROBOT
74    LDD>    D345 K100  ; DATA CHECK SIZE G/T  AT ROBOT
      ANDD<=  D345 K130  ; DATA CHECK SIZE G/T  AT ROBOT
      MOV     K12 D110
84    LDD>    D345 K130  ; DATA CHECK SIZE G/T  AT ROBOT
      ANDD<=  D345 K130  ; DATA CHECK SIZE G/T  AT ROBOT
      MOV     K13 D110
94    LDD>    D345 K130  ; DATA CHECK SIZE G/T  AT ROBOT
      ANDD<=  D345 K200  ; DATA CHECK SIZE G/T  AT ROBOT
      MOV     K14 D110
104   LDD>    D345 K200  ; DATA CHECK SIZE G/T  AT ROBOT
      ANDD<=  D345 K350  ; DATA CHECK SIZE G/T  AT ROBOT
      MOV     K17 D110
114   LDD>    D345 K350  ; DATA CHECK SIZE G/T  AT ROBOT
      ANDD<=  D345 K350  ; DATA CHECK SIZE G/T  AT ROBOT
      MOV     K18 D110
124   LDD>    D345 K350  ; DATA CHECK SIZE G/T  AT ROBOT
      ANDD<=  D345 K360  ; DATA CHECK SIZE G/T  AT ROBOT
      MOV     K19 D110
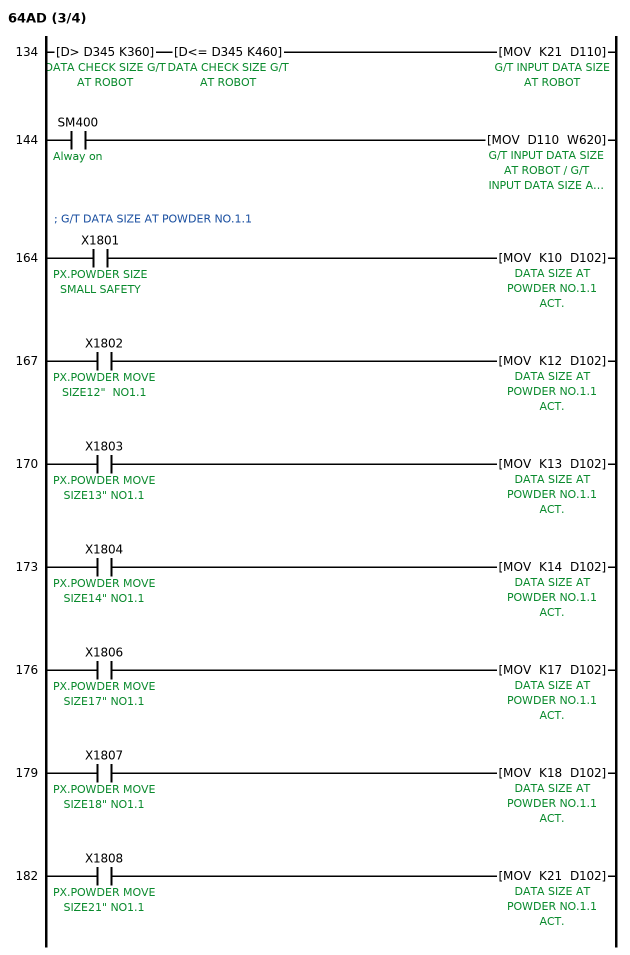
134   LDD>    D345 K360  ; DATA CHECK SIZE G/T  AT ROBOT
      ANDD<=  D345 K460  ; DATA CHECK SIZE G/T  AT ROBOT
      MOV     K21 D110
144   LD      SM400  ; Alway on
      MOV     D110 W620  ; G/T INPUT DATA SIZE AT ROBOT
; G/T DATA SIZE AT POWDER NO.1.1
164   LD      X1801  ; PX.POWDER SIZE SMALL SAFETY
      MOV     K10 D102  ; DATA SIZE AT POWDER NO.1.1 ACT.
167   LD      X1802  ; PX.POWDER MOVE  SIZE12"  NO1.1
      MOV     K12 D102
170   LD      X1803  ; PX.POWDER MOVE SIZE13" NO1.1
      MOV     K13 D102
173   LD      X1804  ; PX.POWDER MOVE SIZE14" NO1.1
      MOV     K14 D102
176   LD      X1806  ; PX.POWDER MOVE SIZE17" NO1.1
      MOV     K17 D102
179   LD      X1807  ; PX.POWDER MOVE SIZE18" NO1.1
      MOV     K18 D102
182   LD      X1808  ; PX.POWDER MOVE SIZE21" NO1.1
      MOV     K21 D102
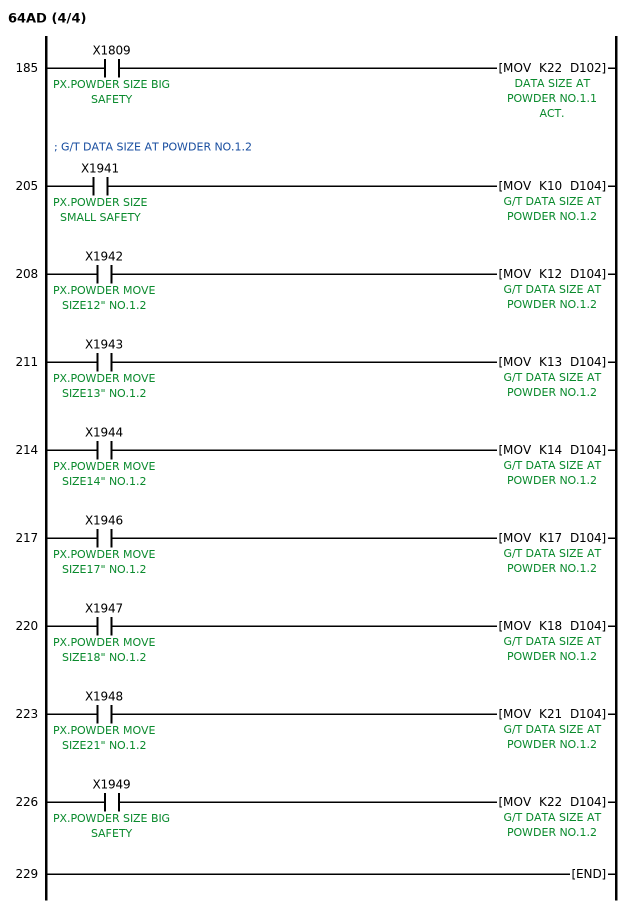
185   LD      X1809  ; PX.POWDER SIZE BIG SAFETY
      MOV     K22 D102
; G/T DATA SIZE AT POWDER NO.1.2
205   LD      X1941  ; PX.POWDER SIZE SMALL SAFETY
      MOV     K10 D104  ; G/T DATA SIZE AT POWDER NO.1.2
208   LD      X1942  ; PX.POWDER MOVE SIZE12" NO.1.2
      MOV     K12 D104
211   LD      X1943  ; PX.POWDER MOVE SIZE13" NO.1.2
      MOV     K13 D104
214   LD      X1944  ; PX.POWDER MOVE SIZE14" NO.1.2
      MOV     K14 D104
217   LD      X1946  ; PX.POWDER MOVE SIZE17" NO.1.2
      MOV     K17 D104
220   LD      X1947  ; PX.POWDER MOVE SIZE18" NO.1.2
      MOV     K18 D104
223   LD      X1948  ; PX.POWDER MOVE SIZE21" NO.1.2
      MOV     K21 D104
226   LD      X1949  ; PX.POWDER SIZE BIG SAFETY
      MOV     K22 D104
229   END
END_PROGRAM

PROGRAM SERVO
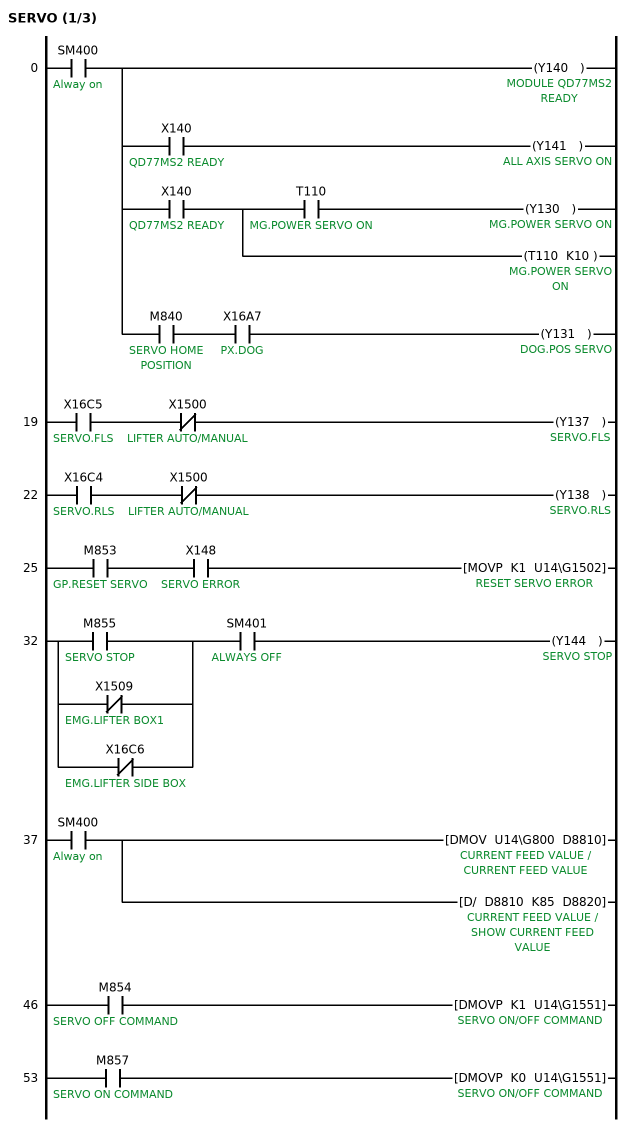
0     LD      SM400  ; Alway on
      OUT     Y140  ; MODULE QD77MS2 READY
      MPS
      AND     X140  ; QD77MS2 READY
      OUT     Y141  ; ALL AXIS SERVO ON
      MRD
      AND     X140  ; QD77MS2 READY
      MPS
      AND     T110  ; MG.POWER SERVO ON
      OUT     Y130  ; MG.POWER SERVO ON
      MPP
      OUT     T110 K10  ; MG.POWER SERVO ON
      MPP
      AND     M840  ; SERVO HOME POSITION
      AND     X16A7  ; PX.DOG
      OUT     Y131  ; DOG.POS SERVO
19    LD      X16C5  ; SERVO.FLS
      ANI     X1500  ; LIFTER AUTO/MANUAL
      OUT     Y137  ; SERVO.FLS
22    LD      X16C4  ; SERVO.RLS
      ANI     X1500  ; LIFTER AUTO/MANUAL
      OUT     Y138  ; SERVO.RLS
25    LD      M853  ; GP.RESET SERVO
      AND     X148  ; SERVO ERROR
      MOVP    K1 U14\G1502  ; RESET SERVO ERROR
32    LD      M855  ; SERVO STOP
      ORI     X1509  ; EMG.LIFTER BOX1
      ORI     X16C6  ; EMG.LIFTER SIDE BOX
      AND     SM401  ; ALWAYS OFF
      OUT     Y144  ; SERVO STOP
37    LD      SM400  ; Alway on
      DMOV    U14\G800 D8810  ; CURRENT FEED VALUE / CURRENT FEED VALUE
      D/      D8810 K85 D8820  ; SHOW CURRENT FEED VALUE
46    LD      M854  ; SERVO OFF COMMAND
      DMOVP   K1 U14\G1551  ; SERVO ON/OFF COMMAND
53    LD      M857  ; SERVO ON COMMAND
      DMOVP   K0 U14\G1551
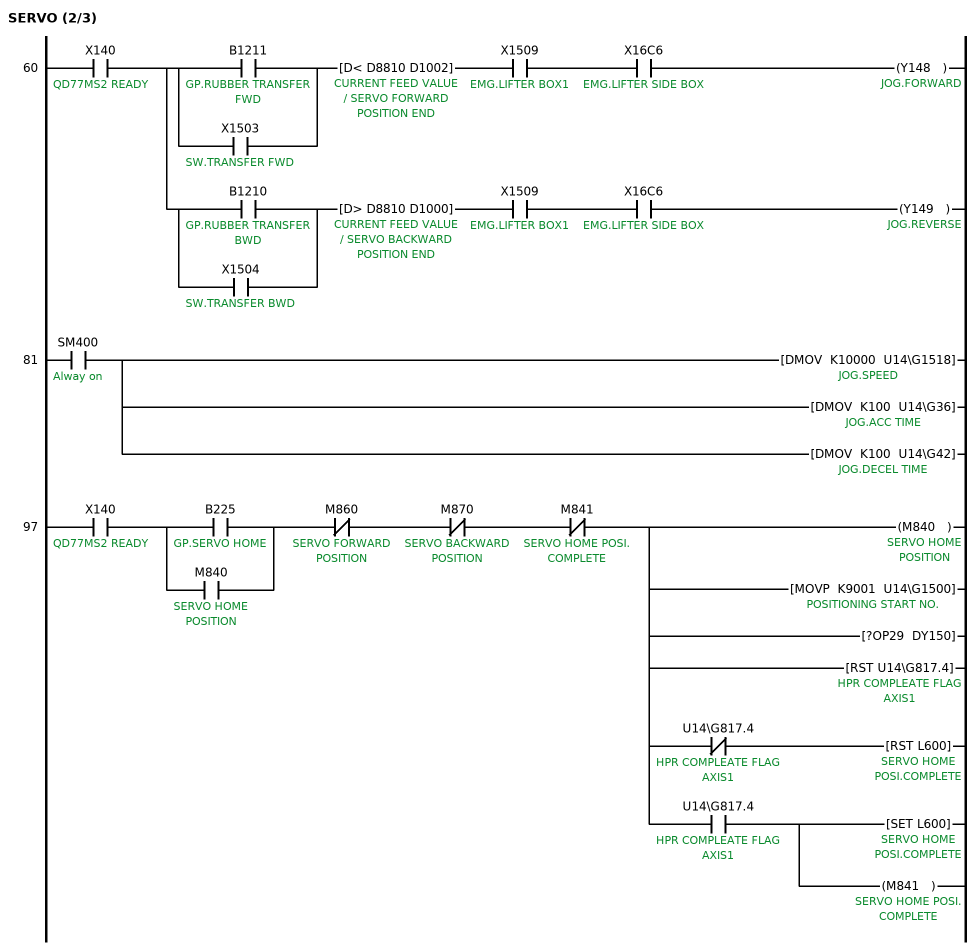
60    LD      X140  ; QD77MS2 READY
      MPS
      LD      B1211  ; GP.RUBBER TRANSFER FWD
      OR      X1503  ; SW.TRANSFER FWD
      ANB
      ANDD<   D8810 D1002  ; CURRENT FEED VALUE / SERVO FORWARD POSITION END
      AND     X1509  ; EMG.LIFTER BOX1
      AND     X16C6  ; EMG.LIFTER SIDE BOX
      OUT     Y148  ; JOG.FORWARD
      MPP
      LD      B1210  ; GP.RUBBER TRANSFER BWD
      OR      X1504  ; SW.TRANSFER BWD
      ANB
      ANDD>   D8810 D1000  ; CURRENT FEED VALUE / SERVO BACKWARD POSITION END
      AND     X1509  ; EMG.LIFTER BOX1
      AND     X16C6  ; EMG.LIFTER SIDE BOX
      OUT     Y149  ; JOG.REVERSE
81    LD      SM400  ; Alway on
      DMOV    K10000 U14\G1518  ; JOG.SPEED
      DMOV    K100 U14\G36  ; JOG.ACC TIME
      DMOV    K100 U14\G42  ; JOG.DECEL TIME
97    LD      X140  ; QD77MS2 READY
      LD      B225  ; GP.SERVO HOME
      OR      M840  ; SERVO HOME POSITION
      ANB
      ANI     M860  ; SERVO FORWARD POSITION
      ANI     M870  ; SERVO BACKWARD POSITION
      ANI     M841  ; SERVO HOME POSI. COMPLETE
      OUT     M840  ; SERVO HOME POSITION
      MOVP    K9001 U14\G1500  ; POSITIONING START NO.
      ?OP29   DY150
      RST     U14\G817.4  ; HPR COMPLEATE FLAG AXIS1
      MPS
      ANI     U14\G817.4  ; HPR COMPLEATE FLAG AXIS1
      RST     L600  ; SERVO HOME POSI.COMPLETE
      MPP
      AND     U14\G817.4  ; HPR COMPLEATE FLAG AXIS1
      SET     L600  ; SERVO HOME POSI.COMPLETE
      OUT     M841  ; SERVO HOME POSI. COMPLETE
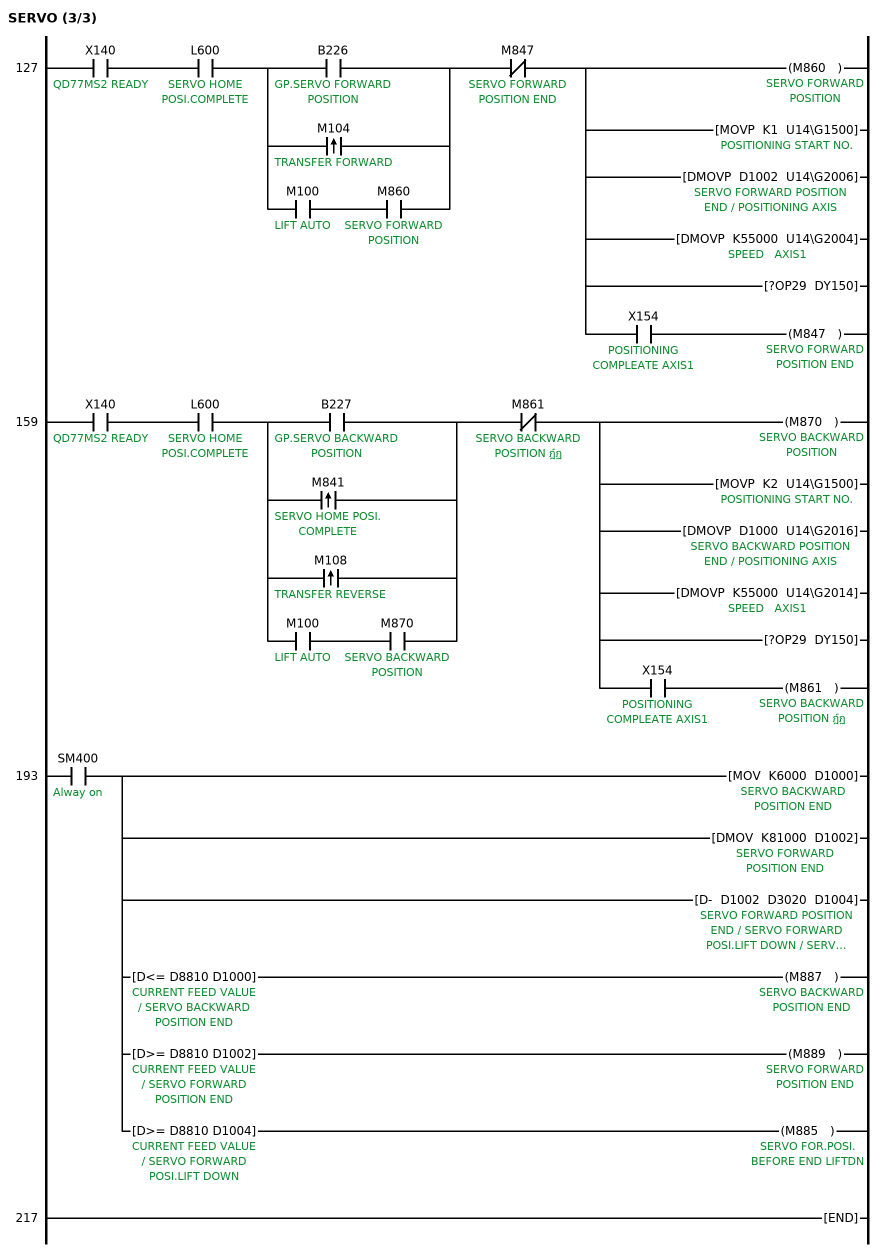
127   LD      X140  ; QD77MS2 READY
      AND     L600  ; SERVO HOME POSI.COMPLETE
      LD      B226  ; GP.SERVO FORWARD POSITION
      ORP     M104  ; TRANSFER FORWARD
      LD      M100  ; LIFT AUTO
      AND     M860  ; SERVO FORWARD POSITION
      ORB
      ANB
      ANI     M847  ; SERVO FORWARD POSITION END
      OUT     M860  ; SERVO FORWARD POSITION
      MOVP    K1 U14\G1500
      DMOVP   D1002 U14\G2006  ; POSITIONING AXIS
      DMOVP   K55000 U14\G2004  ; SPEED   AXIS1
      ?OP29   DY150
      AND     X154  ; POSITIONING COMPLEATE AXIS1
      OUT     M847  ; SERVO FORWARD POSITION END
159   LD      X140  ; QD77MS2 READY
      AND     L600  ; SERVO HOME POSI.COMPLETE
      LD      B227  ; GP.SERVO BACKWARD POSITION
      ORP     M841  ; SERVO HOME POSI. COMPLETE
      ORP     M108  ; TRANSFER REVERSE
      LD      M100  ; LIFT AUTO
      AND     M870  ; SERVO BACKWARD POSITION
      ORB
      ANB
      ANI     M861  ; SERVO BACKWARD POSITION ฎ์ฏ
      OUT     M870  ; SERVO BACKWARD POSITION
      MOVP    K2 U14\G1500
      DMOVP   D1000 U14\G2016  ; POSITIONING AXIS
      DMOVP   K55000 U14\G2014  ; SPEED   AXIS1
      ?OP29   DY150
      AND     X154  ; POSITIONING COMPLEATE AXIS1
      OUT     M861  ; SERVO BACKWARD POSITION ฎ์ฏ
193   LD      SM400  ; Alway on
      MOV     K6000 D1000
      DMOV    K81000 D1002
      D-      D1002 D3020 D1004  ; SERVO FORWARD POSI.LIFT DOWN / SERVO FORWARD POSI.LIFT DOWN
      MPS
      ANDD<=  D8810 D1000  ; CURRENT FEED VALUE / SERVO BACKWARD POSITION END
      OUT     M887  ; SERVO BACKWARD POSITION END
      MRD
      ANDD>=  D8810 D1002  ; CURRENT FEED VALUE / SERVO FORWARD POSITION END
      OUT     M889  ; SERVO FORWARD POSITION END
      MPP
      ANDD>=  D8810 D1004  ; CURRENT FEED VALUE / SERVO FORWARD POSI.LIFT DOWN
      OUT     M885  ; SERVO FOR.POSI.BEFORE END LIFTDN
217   END
END_PROGRAM

PROGRAM D62
